// TIA Portal V19 export
TYPE "ValveMachine_Cin"
// stored: Access Published
   STRUCT
      Manager { S7_SetPoint := 'True'} : "ValveMachine_Manager";
      PressureRunning : Bool;
      Rest_ExtEnable : Bool := TRUE;
      Work_ExtEnable : Bool := TRUE;
      ExternalAlarms : Bool := FALSE;
   END_STRUCT;
END_TYPE
